
// ===== library: MasterCopy "LSim_AllPass1OrdReal" =====

FUNCTION_BLOCK "LSim_AllPass1OrdReal"   // FB61, SCL
{ S7_Optimized_Access := 'TRUE' }
VERSION : 2.01
   VAR_INPUT
      calcParam : Bool;   // recalculate with new parameters
      input : Real;   // input signal
      tmLag1 : Real := 2.0;   // time constant T1 [sec]
      gain : Real := 1.0;   // gain factor
      cycle : Real := 0.1;   // cyclic time [sec]
      maxOut : Real := 100.0;   // max. output limit
      minOut : Real;   // min. output limit
      reset : Bool;   // resets all relevant parameters to ‘0’ including the output
   END_VAR
   VAR_OUTPUT
      error : Bool;   // error (#tmLag1 <= 0)
      status : Word;   // status (if #tmLag1 <= 0 then status = 16#8001)
      maxReached : Bool;   // output has reached max. limit
      minReached : Bool;   // output has reached min. limit
      output : Real;   // output signal (if #error = FALSE)
   END_VAR
   VAR
      statRxn1 : Real;   // delayed input signal (n-1)
      statRyn1 : Real;   // delayed output signal (n-1)
      statRb1 : Real;
      statRa1 : Real;
      statOutput : Real;   // output signal
   END_VAR
BEGIN
   //=============================================================================
   //SIEMENS AG
   //(c)Copyright 2017 All Rights Reserved
   //-----------------------------------------------------------------------------
   //Library:       Library for Controlled System Simulation
   //Tested with:   S7-1500 FW V2.0 / S7-1200 FW V4.2
   //Engineering:   STEP 7 V14 Upd2 (TIA Portal)
   //Restrictions:  Cyclic interrupt
   //Requirements:  memory card needed for S7-1500
   //Functionality: Simulation of an All-Pass 1. Order with real p-Poles
   //
   //         gain * (1 - tmLag1*p)
   //  F(p) = ---------------------
   //            (1 + tmLag1*p)
   //          
   //  Call the simulation in a cyclic interrupt with
   //  cyclic interrupt time at least = tmLag1/10!
   //-----------------------------------------------------------------------------
   //Change log table:
   //Version  Date       Expert in charge                Changes applied
   //02.00.00 03.02.2016 Siemens Industry Online Support Release (STEP 7 V13 SP1)
   //02.00.01 02.03.2017 Siemens Industry Online Support Release (STEP 7 V14)
   //=============================================================================

   // check of the parameter
   IF #tmLag1 <= 0 THEN
     #error := True;
     #status := W#16#8001;     // Parameter Error
     #statRxn1 := 0.0;
     #statRyn1 := 0.0;
     #statOutput := 0;
     #output := 0;
     RETURN;
   ELSE
     #error := FALSE;
     #status := W#16#0000;     // no error
   END_IF;


   // Z-parameters 
   IF #calcParam = True THEN
   // Calculate z-parameters for allpass filter
      #statRa1 := -EXP(-#cycle/#tmLag1);
      #statRb1 := #gain*(2 + #statRa1);

   END_IF;
   // reset Memory
   IF #reset = True THEN
     #statRxn1 := 0.0;
     #statRyn1 := 0.0;
     #statOutput:=0;
     #error := False;
     #status := W#16#0000;
   END_IF;

   // save delayed output signal 
   #statRyn1:= #statOutput;

   // Differencial Equation of all-pass filter 1. order
   #statOutput := #input * (-#gain) +  #statRxn1* #statRb1 - #statRyn1*#statRa1;

   // save delayed input signals
   #statRxn1 := #input;

   // max limit of acutating variable
   IF #statOutput > #maxOut THEN
     #statOutput := #maxOut;
     #maxReached:= True;
   ELSE
     #maxReached := False;
   END_IF;

   // min limit of acutating variable
   IF #statOutput < #minOut THEN
     #statOutput := #minOut;
     #minReached := True;
   ELSE
     #minReached := False;
   END_IF;

   #output := #statOutput;
END_FUNCTION_BLOCK

// ===== library: MasterCopy "LSim_AllPass2OrdReal" =====

FUNCTION_BLOCK "LSim_AllPass2OrdReal"   // FB62, SCL
{ S7_Optimized_Access := 'TRUE' }
VERSION : 2.01
   VAR_INPUT
      calcParam : Bool;   // recalculate with new parameters
      input : Real;   // input signal
      tmLag1 : Real := 2.0;   // time constant T1 [sec]
      tmLag2 : Real := 0.2;   // time constant T2 [sec]
      gain : Real := 1.0;   // gain factor
      cycle : Real := 0.1;   // cyclic time [sec]
      maxOut : Real := 100.0;   // max. output limit
      minOut : Real;   // min. output limit
      reset : Bool;   // resets all relevant parameters to ‘0’ including the output
   END_VAR
   VAR_OUTPUT
      error : Bool;   // error (#tmLag1 <= 0 or #tmLag2 <= 0 or #tmLag2 = #tmLag1)
      status : Word;   // status (if #error = TRUE then status = 16#8001)
      maxReached : Bool;   // output has reached max. limit
      minReached : Bool;   // output has reached min. limit
      output : Real;   // output signal (if #error = FALSE)
   END_VAR
   VAR
      statRxn2 : Real;   // delayed input signal (n-2)
      statRxn1 : Real;   // delayed input signal (n-1)
      statRyn2 : Real;   // delayed output signal (n-2)
      statRyn1 : Real;   // delayed output signal (n-1)
      statRb1 : Real;
      statRb2 : Real;
      statRa1 : Real;
      statRa2 : Real;
      statRe1 : Real;
      statRe2 : Real;
      statRk1 : Real;
      statOverfirst : Bool;
      statOutput : Real;   // output signal
   END_VAR
BEGIN
   //=============================================================================
   //SIEMENS AG
   //(c)Copyright 2017 All Rights Reserved
   //-----------------------------------------------------------------------------
   //Library:       Library for Controlled System Simulation
   //Tested with:   S7-1500 FW V2.0 / S7-1200 FW V4.2
   //Engineering:   STEP 7 V14 Upd2 (TIA Portal)
   //Restrictions:  Cyclic interrupt
   //Requirements:  memory card needed for S7-1500
   //Functionality: Simulation of an All-Pass 2. Order with real p-Poles
   //
   //         gain * (1 - tmLag1*p) * (1 - tmLag2*p)
   //  F(p) = --------------------------------------
   //            (1 + tmLag1*p) * (1 + tmLag2*p)
   //          
   //  Call the simulation in a cyclic interrupt with
   //  cyclic interrupt time at least = tmLag1/10!
   //-----------------------------------------------------------------------------
   //Change log table:
   //Version  Date       Expert in charge                Changes applied
   //02.00.00 03.02.2016 Siemens Industry Online Support Release (STEP 7 V13 SP1)
   //02.00.01 02.03.2017 Siemens Industry Online Support Release (STEP 7 V14)
   //=============================================================================

   // check of the parameter
   IF #tmLag1 <= 0 OR #tmLag2 <= 0 OR #tmLag1 = #tmLag2 THEN
     #error := TRUE;
     #status := W#16#8001;     // Parameter Error
     #statRxn1 := 0.0;
     #statRyn1 := 0.0;
     #statRxn2 := 0.0;
     #statRyn2 := 0.0;
     #statOutput := 0;
     #output := 0;
     RETURN;
   ELSE
     #error := FALSE;
     #status := W#16#0000;     // no error
   END_IF;

   // calculates the z-parameter for the difference equatation
   IF #calcParam = True OR NOT #statOverfirst THEN
   // Calculate z-parameters for oscilating PT2-System
   #statOverfirst:=1;
   #statRe1 := -EXP(-#cycle/#tmLag1);
   #statRe2 := -EXP(-#cycle/#tmLag2);
   #statRk1 := (2* (#tmLag2 + #tmLag1))/(#tmLag2 - #tmLag1);
   #statRa1 := #statRe1 + #statRe2;
   #statRa2 := #statRe1*#statRe2;
   #statRb1 := #gain*(#statRa1+ #statRk1*(#statRe2 - #statRe1));
   #statRb2 := #gain*(#statRa2 -#statRk1*(#statRe2 - #statRe1));
   END_IF;

   // reset memory
   IF #reset = True THEN
     #statRxn1 := 0.0;
     #statRyn1 := 0.0;
     #statRxn2 := 0.0;
     #statRyn2 := 0.0;
     #statOutput:=0;
     #error := False;
     #status := W#16#0000;
   END_IF;

   // save delayed output-signals
   #statRyn2:=#statRyn1;
   #statRyn1:= #statOutput;

   // difference equatation for PT2-system
   #statOutput := #input * #gain +  #statRxn1* #statRb1 + #statRxn2*#statRb2 - #statRyn1*#statRa1 - #statRyn2*#statRa2;

   // save delayed input-signals
   #statRxn2 := #statRxn1;
   #statRxn1 := #input;

   // max limit of acutating variable
   IF #statOutput > #maxOut THEN
     #statOutput := #maxOut;
     #maxReached:= True;
   ELSE
     #maxReached := False;
   END_IF;

   // min limit of acutating variable
   IF #statOutput < #minOut THEN
     #statOutput := #minOut;
     #minReached := True;
   ELSE
     #minReached := False;
   END_IF;

   #output := #statOutput;
END_FUNCTION_BLOCK

// ===== library: MasterCopy "LSim_DT1" =====

FUNCTION_BLOCK "LSim_DT1"   // FB60, SCL
{ S7_Optimized_Access := 'TRUE' }
VERSION : 2.01
   VAR_INPUT
      calcParam : Bool;   // recalculate with new parameters
      input : Real;   // input signal
      tmLag1 : Real := 2.0;   // time constant T1 [sec]
      tmLag2 : Real := 0.5;   // time constant T2 [sec]
      gain : Real := 1.0;   // gain factor
      cycle : Real := 0.1;   // cyclic time [sec]
      maxOut : Real := 100.0;   // max. output limit
      minOut : Real := -100.0;   // min. output limit
      reset : Bool;   // resets all relevant parameters to ‘0’ including the output
   END_VAR
   VAR_OUTPUT
      error : Bool;   // error (#tmLag1 <= 0)
      status : Word;   // status (if #tmLag1 <= 0 then status = 16#8001)
      maxReached : Bool;   // output has reached max. limit
      minReached : Bool;   // output has reached min. limit
      output : Real;   // output signal (if #error = FALSE)
   END_VAR
   VAR
      statRxn1 : Real;   // delayed input signal (n-1)
      statRyn1 : Real;   // delayed output signal (n-1)
      statRb0 : Real;
      statRa1 : Real;
      statOverfirst : Bool;
      statOutput : Real;   // output signal
   END_VAR
BEGIN
   //=============================================================================
   //SIEMENS AG
   //(c)Copyright 2017 All Rights Reserved
   //-----------------------------------------------------------------------------
   //Library:       Library for Controlled System Simulation
   //Tested with:   S7-1500 FW V2.0 / S7-1200 FW V4.2
   //Engineering:   STEP 7 V14 Upd2 (TIA Portal)
   //Restrictions:  Cyclic interrupt
   //Requirements:  memory card needed for S7-1500
   //Functionality: Simulation of a DT1-System
   //
   //         gain * tmLag2 * p
   //  F(p) = ------------------------------
   //            (1 + tmLag1*p)
   //          
   //  Call the simulation in a cyclic interrupt with
   //  cyclic interrupt time at least = tmLag1/10!
   //-----------------------------------------------------------------------------
   //Change log table:
   //Version  Date       Expert in charge                Changes applied
   //02.00.00 03.02.2016 Siemens Industry Online Support Release (STEP 7 V13 SP1)
   //02.00.01 02.03.2017 Siemens Industry Online Support Release (STEP 7 V14)
   //=============================================================================

   // check of the parameter
   IF #tmLag1 <= 0 THEN
     #error := true;
     #status := W#16#8001; // parameter error
     #statRxn1 := 0.0;
     #statRyn1 := 0.0;
     #statOutput := 0;
     #output := 0;
     RETURN;
   ELSE
     #error := FALSE;
     #status := W#16#0000;     // no error
   END_IF;

   // calculates the z-parameter for the difference equatation
   IF #calcParam = True OR NOT #statOverfirst THEN 
     // Calculate the z-parameter for the DT1-System
     #statOverfirst := 1;
     #statRa1 := -EXP(-#cycle/#tmLag1);
     #statRb0 := #gain*(#tmLag2/#tmLag1);
   END_IF;

   // reset Memory
   IF #reset = True THEN
     #statRxn1 := 0.0;
     #statRyn1 := 0.0;
     #statOutput:=0;
     #error := false;
     #status := W#16#0000;
   END_IF;

   // save delayed output-signals
   #statRyn1:= #statOutput;

   //  difference equatation for DT1-system
   #statOutput := #input * #statRb0 - #statRxn1* #statRb0 - #statRyn1*#statRa1;

   // save delayed input-signals
   #statRxn1 := #input;

   // max limit of acutating variable
   IF #statOutput > #maxOut THEN
     #statOutput := #maxOut;
     #maxReached := True;
   ELSE
     #maxReached := False;
   END_IF;

   // min limit of acutating variable
   IF #statOutput < #minOut THEN
     #statOutput := #minOut;
     #minReached := True;
   ELSE
     #minReached := False;
   END_IF;

   #output := #statOutput;
END_FUNCTION_BLOCK

// ===== library: MasterCopy "LSim_I" =====

FUNCTION_BLOCK "LSim_I"   // FB56, SCL
{ S7_Optimized_Access := 'TRUE' }
VERSION : 2.01
   VAR_INPUT
      calcParam : Bool;   // recalculate with new parameters
      input : Real;   // input signal
      tmLag1 : Real := 1.0;   // time constant T1 [sec]
      cycle : Real := 0.1;   // cyclic time [sec]
      maxOut : Real := 100.0;   // max. output limit
      minOut : Real;   // min. output limit
      reset : Bool;   // resets all relevant parameters to ‘0’ including the output
   END_VAR
   VAR_OUTPUT
      error : Bool;   // error (#tmLag1 <= 0)
      status : Word;   // status (if #tmLag1 <= 0 then status = 16#8001)
      maxReached : Bool;   // output has reached max. limit
      minReached : Bool;   // output has reached min. limit
      output : Real;   // output signal (if #error = FALSE)
   END_VAR
   VAR
      statRxn1 : Real;   // delayed input signal (n-1)
      statRyn1 : Real;   // delayed output signal (n-1)
      statRa1 : Real;
      statRb1 : Real;
      statOverfirst : Bool;
      statOutput : Real;   // output signal
   END_VAR
BEGIN
   //=============================================================================
   //SIEMENS AG
   //(c)Copyright 2017 All Rights Reserved
   //-----------------------------------------------------------------------------
   //Library:       Library for Controlled System Simulation
   //Tested with:   S7-1500 FW V2.0 / S7-1200 FW V4.2
   //Engineering:   STEP 7 V14 Upd2 (TIA Portal)
   //Restrictions:  Cyclic interrupt
   //Requirements:  memory card needed for S7-1500
   //Functionality: Simulation of a I-System
   //
   //             1
   //  F(p) = -----------
   //         (tmLag1*p)
   //          
   //  Call the simulation in a cyclic interrupt with
   //  cyclic interrupt time at least = tmLag1/10!
   //-----------------------------------------------------------------------------
   //Change log table:
   //Version  Date       Expert in charge                Changes applied
   //02.00.00 03.02.2016 Siemens Industry Online Support Release (STEP 7 V13 SP1)
   //02.00.01 02.03.2017 Siemens Industry Online Support Release (STEP 7 V14)
   //=============================================================================

   // check parameter
   IF #tmLag1 <= 0 THEN
     #error := True;
     #status := W#16#8001;     // Parameter Error
     #statRxn1 := 0.0;
     #statRyn1 := 0.0;
     #statOutput := 0;
     #output := 0;
     RETURN;
   ELSE
     #error := FALSE;
     #status := W#16#0000;     // no error
   END_IF;

   // calculates the z-parameter for the difference equatation
   IF #calcParam = True OR NOT #statOverfirst THEN
   #statOverfirst:=1;
     // Calculate z-parameters for IT1-System
   #statRb1 := #cycle/#tmLag1;
   #statRa1 := -1;

   END_IF;

   // reset Memory
   IF #reset = True THEN
     #statRxn1 := 0.0;
     #statRyn1 := 0.0;
     #statOutput:=0;
   END_IF;

   // save delayed output-signals
   #statRyn1:= #statOutput;

   // difference equatation for the I-system
   #statOutput := #statRxn1* #statRb1 - #statRyn1*#statRa1;

   // save delayed input-signals
   #statRxn1 := #input;

   // max limit of acutating variable
   IF #statOutput > #maxOut THEN
     #statOutput := #maxOut;
     #maxReached:= True;
   ELSE
     #maxReached := False;
   END_IF;

   // min limit of acutating variable
   IF #statOutput < #minOut THEN
     #statOutput := #minOut;
     #minReached := True;
   ELSE
     #minReached := False;
   END_IF;

   #output := #statOutput;
END_FUNCTION_BLOCK

// ===== library: MasterCopy "LSim_IT1" =====

FUNCTION_BLOCK "LSim_IT1"   // FB57, SCL
{ S7_Optimized_Access := 'TRUE' }
VERSION : 2.01
   VAR_INPUT
      calcParam : Bool;   // recalculate with new parameters
      input : Real;   // input signal
      tmLag1 : Real := 5.0;   // time constant T1 [sec]
      gain : Real := 1.0;   // gain factor
      cycle : Real := 0.1;   // cyclic time [sec]
      maxOut : Real := 100.0;   // max. output limit
      minOut : Real;   // min. output limit
      reset : Bool;   // resets all relevant parameters to ‘0’ including the output
   END_VAR
   VAR_OUTPUT
      error : Bool;   // error (#tmLag1 <= 0)
      status : Word;   // status (if #tmLag1 <= 0 then status = 16#8001)
      maxReached : Bool;   // output has reached max. limit
      minReached : Bool;   // output has reached min. limit
      output : Real;   // output signal (if #error = FALSE)
   END_VAR
   VAR
      statRxn2 : Real;   // delayed input signal (n-2)
      statRxn1 : Real;   // delayed input signal (n-1)
      statRyn2 : Real;   // delayed output signal (n-2)
      statRyn1 : Real;   // delayed output signal (n-1)
      statRf1 : Real;
      statRf2 : Real;
      statRe1 : Real;
      statRe2 : Real;
      statAlpha : Real;
      statOverfirst : Bool;
      statOutput : Real;   // output signal
   END_VAR
BEGIN
   //=============================================================================
   //SIEMENS AG
   //(c)Copyright 2017 All Rights Reserved
   //-----------------------------------------------------------------------------
   //Library:       Library for Controlled System Simulation
   //Tested with:   S7-1500 FW V2.0 / S7-1200 FW V4.2
   //Engineering:   STEP 7 V14 Upd2 (TIA Portal)
   //Restrictions:  Cyclic interrupt
   //Requirements:  memory card needed for S7-1500
   //Functionality: Simulation of a IT1-System
   //  
   //               gain
   //  F(p) = ------------------
   //         p * (tmLag1*p + 1)
   //         
   //  Call the simulation in a cyclic interrupt with
   //  cyclic interrupt time at least = tmLag1/10!
   //-----------------------------------------------------------------------------
   //Change log table:
   //Version  Date       Expert in charge                Changes applied
   //02.00.00 03.02.2016 Siemens Industry Online Support Release (STEP 7 V13 SP1)
   //02.00.01 02.03.2017 Siemens Industry Online Support Release (STEP 7 V14)
   //=============================================================================


   // check parameter
   IF #tmLag1 <= 0 THEN
     #error := True;
     #status := W#16#8001;     // Parameter Error
     #statRxn1 := 0.0;
     #statRyn1 := 0.0;
     #statRxn2 := 0.0;
     #statRyn2 := 0.0;
     #statOutput := 0;
     #output := 0;
     RETURN;
   ELSE
     #error := FALSE;
     #status := W#16#0000;     // no error
   END_IF;

   // calculates the z-parameter for the difference equatation
   IF #calcParam = True OR NOT #statOverfirst THEN
     #statOverfirst:=1;
   // calculates the z-parameter for the difference equatation of the IT1-System
   #statAlpha := EXP(-#cycle/#tmLag1);
   #statRe1 := -1 - #statAlpha;
   #statRe2 := #statAlpha;
   #statRf1 := #gain*(#cycle +(#statAlpha - 1)*#tmLag1);
   #statRf2 := #gain*(-#statAlpha*#cycle+(1-#statAlpha)*#tmLag1);
   END_IF;

   // reset Memory
   IF #reset = True THEN
     #statRxn1 := 0.0;
     #statRyn1 := 0.0;
     #statRxn2 := 0.0;
     #statRyn2 := 0.0;
     #statOutput:=0;
   END_IF;

   // save delayed output-signals
   #statRyn2:=#statRyn1;
   #statRyn1:= #statOutput;

   // difference equatation for IT1-System
   #statOutput := #statRxn1* #statRf1 + #statRxn2*#statRf2 - #statRyn1*#statRe1 - #statRyn2*#statRe2;

   // save delayed input-signals
   #statRxn2 := #statRxn1;
   #statRxn1 := #input;

   // max limit of acutating variable
   IF #statOutput > #maxOut THEN
   #statOutput := #maxOut;
   #maxReached := True;
   ELSE
     #maxReached := False;
   END_IF;

   // min limit of acutating variable
   IF #statOutput < #minOut THEN
     #statOutput := #minOut;
     #minReached := True;
   ELSE
     #minReached := False;
   END_IF;

   #output := #statOutput;
END_FUNCTION_BLOCK

// ===== library: MasterCopy "LSim_Lagging" =====

FUNCTION_BLOCK "LSim_Lagging"   // FB59, SCL
{ S7_Optimized_Access := 'TRUE' }
VERSION : 2.02
   VAR_INPUT
      input : Real;   // input signal
   END_VAR
   VAR_OUTPUT
      output : Real;   // output signal
   END_VAR
   VAR_IN_OUT
      delayCycles : UInt;   // number of cycles the input signal is delayed (if #delayCycles > #MAX then #delayCycles = #MAX)
   END_VAR
   VAR
      statDelayStore : Array[0..#MAX] of Real;
      statIndexRead : Int;
      statIndexWrite : Int;
   END_VAR
   VAR CONSTANT
      MAX : Int := 100;   // maximum size of array #statDelayStore
   END_VAR
BEGIN
   //=============================================================================
   //SIEMENS AG
   //(c)Copyright 2017 All Rights Reserved
   //-----------------------------------------------------------------------------
   //Library:       Library for Controlled System Simulation
   //Tested with:   S7-1500 FW V2.0 / S7-1200 FW V4.2
   //Engineering:   STEP 7 V14 Upd2 (TIA Portal)
   //Restrictions:  Cyclic interrupt
   //Requirements:  memory card needed for S7-1500
   //Functionality: Simulation of an Tt-System (Lagging)
   //
   //  F(p) = EXP(-p * delayCycles * cyclic interrupt time)
   //          
   //  Call the simulation in a cyclic interrupt with
   //  cyclic interrupt time at least = tmLag1/10!
   //-----------------------------------------------------------------------------
   //Change log table:
   //Version  Date       Expert in charge                Changes applied
   //02.00.00 03.02.2016 Siemens Industry Online Support Release (STEP 7 V13 SP1)
   //02.00.01 02.03.2017 Siemens Industry Online Support Optimize program code
   //02.00.02 02.03.2017 Siemens Industry Online Support Release (STEP 7 V14)
   //=============================================================================

   // Check Parameters
   IF #delayCycles > #MAX THEN
     #delayCycles := INT_TO_UINT(#MAX);
   ELSE
     #delayCycles := #delayCycles;
   END_IF;

   IF #statIndexWrite < #delayCycles THEN
     #statDelayStore[#statIndexWrite] := #input;   // write input at delayStore indexWrite
     #statIndexRead := #statIndexWrite + 1;
     #output := #statDelayStore[#statIndexRead];   // read output from delayStore indexWrite + 1
     #statIndexWrite := #statIndexWrite + 1;       // increment delayStore indexWrite
   ELSE // maximum reached
     #statDelayStore[#statIndexWrite] := #input;   // write input at delayStore maximum
     #statIndexRead := 0;                          // set indexRead to beginning
     #output := #statDelayStore[#statIndexRead];   // read output from delayStore indexRead
     #statIndexWrite := 0;                         // set indexWrite to beginning
   END_IF;
END_FUNCTION_BLOCK

// ===== library: MasterCopy "LSim_PDT1" =====

FUNCTION_BLOCK "LSim_PDT1"   // FB55, SCL
{ S7_Optimized_Access := 'TRUE' }
VERSION : 2.01
   VAR_INPUT
      calcParam : Bool;   // recalculate with new parameters
      input : Real;   // input signal
      tmLag1 : Real := 2.0;   // time constant T1 [sec]
      tmLag2 : Real := 0.2;   // time constant T2 [sec]
      gain : Real := 1.0;   // gain factor
      cycle : Real := 0.1;   // cyclic time [sec]
      maxOut : Real := 100.0;   // max. output limit
      minOut : Real;   // min. output limit
      reset : Bool;   // resets all relevant parameters to ‘0’ including the output
   END_VAR
   VAR_OUTPUT
      error : Bool;   // error (#tmLag1 <= 0 or #tmLag2 <= 0)
      status : Word;   // status (if #error = TRUE then status = 16#8001)
      maxReached : Bool;   // output has reached max. limit
      minReached : Bool;   // output has reached min. limit
      output : Real;   // output signal (if #error = FALSE)
   END_VAR
   VAR
      statRxn2 : Real;   // delayed input signal (n-2)
      statRxn1 : Real;   // delayed input signal (n-1)
      statRyn2 : Real;   // delayed output signal (n-2)
      statRyn1 : Real;   // delayed output signal (n-1)
      statRb1 : Real;
      statRb0 : Real;
      statRa1 : Real;
      statOverfirst : Bool;
      statOutput : Real;
   END_VAR
BEGIN
   //=============================================================================
   //SIEMENS AG
   //(c)Copyright 2017 All Rights Reserved
   //-----------------------------------------------------------------------------
   //Library:       Library for Controlled System Simulation
   //Tested with:   S7-1500 FW V2.0 / S7-1200 FW V4.2
   //Engineering:   STEP 7 V14 Upd2 (TIA Portal)
   //Restrictions:  Cyclic interrupt
   //Requirements:  memory card needed for S7-1500
   //Functionality: Simulation of an PD-T1 System
   //
   //         gain * (1 + tmLag2*p)
   //  F(p) = ------------------------------
   //            (1 + tmLag1*p)
   //          
   //  Call the simulation in a cyclic interrupt with
   //  cyclic interrupt time at least = tmLag1/10!
   //-----------------------------------------------------------------------------
   //Change log table:
   //Version  Date       Expert in charge                Changes applied
   //02.00.00 03.02.2016 Siemens Industry Online Support Release (STEP 7 V13 SP1)
   //02.00.01 02.03.2017 Siemens Industry Online Support Release (STEP 7 V14)
   //=============================================================================

   // check parameter
   IF #tmLag1 <= 0 OR #tmLag2 <= 0 THEN
     #error := True;
     #status := W#16#8001;     // Parameter Error
     #statRxn1 := 0.0;
     #statRyn1 := 0.0;
     #statRxn2 := 0.0;
     #statRyn2 := 0.0;
     #statOutput := 0;
     #output := 0;
     RETURN;
   ELSE
     #error := FALSE;
     #status := W#16#0000;     // no error
   END_IF;

   // calculates the z-parameter for the difference equatation
   IF #calcParam = True OR NOT #statOverfirst THEN
     #statOverfirst := 1;
   // Calculate z-parameters for oscilating PT2-System
   #statRa1 := -EXP(-#cycle/#tmLag1);
   #statRb0 := #gain *(#tmLag2/#tmLag1);
   #statRb1 := #gain *(1 + #statRa1 - (#tmLag2/#tmLag1));
   END_IF;

   // reset Memory
   IF #reset = True THEN
     #statRxn1 := 0.0;
     #statRyn1 := 0.0;
     #statRxn2 := 0.0;
     #statRyn2 := 0.0;
     #statOutput:=0;
     #error := False;
     #status := W#16#0000;
   END_IF;

   // save delayed output-signals
   #statRyn1:= #statOutput;

   // difference equatation for PT2-system
   #statOutput := #input * #statRb0 +  #statRxn1* #statRb1 - #statRyn1*#statRa1;

   // save delayed input-signals
   #statRxn1 := #input;

   // max limit of acutating variable
   IF #statOutput > #maxOut THEN
     #statOutput := #maxOut;
     #maxReached:= True;
   ELSE
     #maxReached := False;
   END_IF;

   // min limit of acutating variable
   IF #statOutput < #minOut THEN
     #statOutput := #minOut;
     #minReached := True;
   ELSE
     #minReached := False;
   END_IF;

   #output := #statOutput;
END_FUNCTION_BLOCK

// ===== library: MasterCopy "LSim_PT1" =====

FUNCTION_BLOCK "LSim_PT1"   // FB50, SCL
{ S7_Optimized_Access := 'TRUE' }
VERSION : 2.01
   VAR_INPUT
      calcParam : Bool;   // recalculate with new parameters
      input : Real;   // input signal
      tmLag1 : Real := 1.0;   // time constant T1 [sec]
      gain : Real := 1.0;   // gain factor
      cycle : Real := 0.1;   // cyclic time [sec]
      maxOut : Real := 100.0;   // max. output limit
      minOut : Real;   // min. output limit
      reset : Bool;   // resets all relevant parameters to ‘0’ including the output
   END_VAR
   VAR_OUTPUT
      error : Bool;   // error (#tmLag1 <= 0)
      status : Word;   // status (if #tmLag1 <= 0 then status = 16#8001)
      maxReached : Bool;   // output has reached max. limit
      minReached : Bool;   // output has reached min. limit
      output : Real;   // output signal (if #error = FALSE)
   END_VAR
   VAR
      statRf1 : Real;
      statRe1 : Real;
      statOverfirst : Bool;
      statOutput : Real;
   END_VAR
BEGIN
   //=============================================================================
   //SIEMENS AG
   //(c)Copyright 2017 All Rights Reserved
   //-----------------------------------------------------------------------------
   //Library:       Library for Controlled System Simulation
   //Tested with:   S7-1500 FW V2.0 / S7-1200 FW V4.2
   //Engineering:   STEP 7 V14 Upd2 (TIA Portal)
   //Restrictions:  Cyclic interrupt
   //Requirements:  memory card needed for S7-1500
   //Functionality: Simulation of a PT1-System
   //
   //              gain
   //  F(p) = ---------------
   //          tmLag1 * p + 1
   //          
   //  Call the simulation in a cyclic interrupt with
   //  cyclic interrupt time at least = tmLag1/10!
   //-----------------------------------------------------------------------------
   //Change log table:
   //Version  Date       Expert in charge                Changes applied
   //02.00.00 03.02.2016 Siemens Industry Online Support Release (STEP 7 V13 SP1)
   //02.00.01 02.03.2017 Siemens Industry Online Support Release (STEP 7 V14)
   //=============================================================================
   // check parameter
   IF #tmLag1 <= 0 THEN
     #error := TRUE;
     #status := W#16#8001;     // Parameter Error
     #statOutput := 0;
     #output := 0;
     RETURN;
   ELSE
     #error := FALSE;
     #status := W#16#0000;     // no error
   END_IF;

   IF #calcParam = True OR NOT #statOverfirst THEN
     #statOverfirst:=1;
   // Z-parameters For Laplace PT1-System
   #statRe1 := - EXP(-#cycle/#tmLag1);
   #statRf1 := #gain*(1 + #statRe1);
   END_IF;

   // Differencial Equation of PT1-System
   #statOutput := #input*#statRf1 - #statOutput*#statRe1;

   // max limit of acutating variable
   IF #statOutput > #maxOut THEN
     #statOutput := #maxOut;
     #maxReached:= True;
   ELSE
     #maxReached := False;
   END_IF;

   // min limit of acutating variable
   IF #statOutput < #minOut THEN
     #statOutput := #minOut;
     #minReached := True;
   ELSE
     #minReached := False;
   END_IF;

   IF #reset THEN
     #statOutput := 0;
   END_IF;

   #output := #statOutput;
END_FUNCTION_BLOCK

// ===== library: MasterCopy "LSim_PT1asym" =====

FUNCTION_BLOCK "LSim_PT1asym"   // FB51, SCL
{ S7_Optimized_Access := 'TRUE' }
VERSION : 2.01
   VAR_INPUT
      calcParam : Bool;   // recalculate with new parameters
      input : Real;   // input signal
      tmLag1up : Real := 1.0;   // time constant T1 [sec] rising input
      tmLag1down : Real := 10.0;   // time constant T1 [sec] falling input
      gain : Real := 1.0;   // gain factor
      cycle : Real := 0.1;   // cyclic time [sec]
      maxOut : Real := 100.0;   // max. output limit
      minOut : Real;   // min. output limit
      reset : Bool;   // resets all relevant parameters to ‘0’ including the output
   END_VAR
   VAR_OUTPUT
      error : Bool;   // error (#tmLag1 <= 0 or #tmLag2 <= 0)
      status : Word;   // status (if #error = TRUE then status = 16#8001)
      maxReached : Bool;   // output has reached max. limit
      minReached : Bool;   // output has reached min. limit
      output : Real;   // output signal (if #error = FALSE)
   END_VAR
   VAR
      statRxn1 : Real;   // delayed input signal (n-1)
      statRyn1 : Real;   // delayed output signal (n-1)
      statRf1up : Real;   // Z-parameter 1 (rising xn)
      statRe1up : Real;   // Z-parameter 2 (rising xn)
      statRf1dn : Real;   // Z-parameter 1 (falling xn)
      statRe1dn : Real;   // Z-parameter 2 (falling xn)
      statRf1 : Real;   // active Z-parameter 1
      statRe1 : Real;   // active Z-parameter 2
      statOverfirst : Bool;
      statOutput : Real;
   END_VAR
BEGIN
   //=============================================================================
   //SIEMENS AG
   //(c)Copyright 2017 All Rights Reserved
   //-----------------------------------------------------------------------------
   //Library:       Library for Controlled System Simulation
   //Tested with:   S7-1500 FW V2.0 / S7-1200 FW V4.2
   //Engineering:   STEP 7 V14 Upd2 (TIA Portal)
   //Restrictions:  Cyclic interrupt
   //Requirements:  memory card needed for S7-1500
   //Functionality: Simulation of a PT1-System with two different Time-Constants
   //
   //  tmLag1up: Time-Constant for positive Inputsignal changes 
   //  tmLag1down: Time-Constant for negative Inputsignal changes
   //  
   //                gain
   //  Fup(p) = ----------------
   //           tmLag1up * p + 1
   //          
   //                    gain
   //  Fdown(p) = ------------------
   //             tmLag1down * p + 1
   //          
   //  Call the simulation in a cyclic interrupt with
   //  //  cyclic interrupt time at least = tmLag1/10!
   //-----------------------------------------------------------------------------
   //Change log table:
   //Version  Date       Expert in charge                Changes applied
   //02.00.00 03.02.2016 Siemens Industry Online Support Release (STEP 7 V13 SP1)
   //02.00.01 02.03.2017 Siemens Industry Online Support Release (STEP 7 V14)
   //=============================================================================

   // check parameter
   IF #tmLag1up <= 0 OR #tmLag1down <= 0 THEN
     #error := TRUE;
     #status := W#16#8001;     // Parameter Error
     #statOutput := 0;
     #output := 0;
     RETURN;
   ELSE
     #error := FALSE;
     #status := W#16#0000;     // no error
   END_IF;

   IF #calcParam = True OR NOT #statOverfirst THEN
     #statOverfirst:=1;
   // Z-parameters for Laplace PT1-System (rising signal change)
   #statRe1up := - EXP(-#cycle/#tmLag1up);
   #statRf1up := #gain*(1 + #statRe1up);
   // Z-parameters for Laplace PT1-System (falling signal change)
   #statRe1dn := - EXP(-#cycle/#tmLag1down);
   #statRf1dn := #gain*(1 + #statRe1dn);
   END_IF;

   // save delayed output signals
   #statRyn1:= #statOutput;

   // Change the parameter sets, dependent to Input Change
   IF (#input - #statRxn1) > 0 THEN
     #statRf1 := #statRf1up;
     #statRe1 := #statRe1up;
   ELSIF (#input - #statRxn1) < 0 THEN
      #statRf1 := #statRf1dn;
      #statRe1 := #statRe1dn;
   ELSE
     ;
   END_IF;

   // Differencial Equation of PT1-System
   #statOutput := #input*#statRf1 - #statRyn1*#statRe1;

   // save delayed input signals
   #statRxn1 := #input;

   // max limit of acutating variable
   IF #statOutput > #maxOut THEN
     #statOutput := #maxOut;
     #maxReached:= True;
   ELSE
     #maxReached := False;
   END_IF;

   // min limit of acutating variable
   IF #statOutput < #minOut THEN
     #statOutput := #minOut;
     #minReached := True;
   ELSE
     #minReached := False;
   END_IF;

   IF #reset THEN
     #statOutput := 0;
   END_IF;

   #output := #statOutput;
END_FUNCTION_BLOCK

// ===== library: MasterCopy "LSim_PT2aper" =====

FUNCTION_BLOCK "LSim_PT2aper"   // FB53, SCL
{ S7_Optimized_Access := 'TRUE' }
VERSION : 2.01
   VAR_INPUT
      calcParam : Bool;   // recalculate with new parameters
      input : Real;   // input signal
      tmLag1 : Real := 2.0;   // time constant T1 [sec]
      tmLag2 : Real := 0.2;   // time constant T2 [sec]
      gain : Real := 1.0;   // gain factor
      cycle : Real := 0.1;   // cyclic time [sec]
      maxOut : Real := 100.0;   // max. output limit
      minOut : Real;   // min. output limit
      reset : Bool;   // resets all relevant parameters to ‘0’ including the output
   END_VAR
   VAR_OUTPUT
      error : Bool;   // error (#tmLag1 <= 0 or #tmLag2 <= 0 or #tmLag1 = #tmLag2)
      status : Word;   // status (if #error = TRUE then status = 16#8001)
      maxReached : Bool;   // output has reached max. limit
      minReached : Bool;   // output has reached min. limit
      output : Real;   // output signal (if #error = FALSE)
   END_VAR
   VAR
      statRxn2 : Real;   // delayed input signal (n-2)
      statRxn1 : Real;   // delayed input signal (n-1)
      statRyn2 : Real;   // delayed output signal (n-2)
      statRyn1 : Real;   // delayed output signal (n-1)
      statRf1 : Real;
      statRf2 : Real;
      statRe1 : Real;
      statRe2 : Real;
      statAlpha : Real;
      statBeta : Real;
      statGamma : Real;
      statDelta : Real;
      statOverfirst : Bool;
      statOutput : Real;   // Output signal
   END_VAR
BEGIN
   //=============================================================================
   //SIEMENS AG
   //(c)Copyright 2017 All Rights Reserved
   //-----------------------------------------------------------------------------
   //Library:       Library for Controlled System Simulation
   //Tested with:   S7-1500 FW V2.0 / S7-1200 FW V4.2
   //Engineering:   STEP 7 V14 Upd2 (TIA Portal)
   //Restrictions:  Cyclic interrupt
   //Requirements:  memory card needed for S7-1500
   //Functionality: Simulation of a aperiodic PT2-System
   //  
   //                    gain
   //  F(p) = -----------------------------
   //         (tmLag1*p + 1)*(tmLag2*p + 1)
   //         
   //  Call the simulation in a cyclic interrupt with
   //  cyclic interrupt time at least = tmLag1/10!
   //-----------------------------------------------------------------------------
   //Change log table:
   //Version  Date       Expert in charge                Changes applied
   //02.00.00 03.02.2016 Siemens Industry Online Support Release (STEP 7 V13 SP1)
   //02.00.01 02.03.2017 Siemens Industry Online Support Release (STEP 7 V14)
   //=============================================================================

   // check parameter
   IF #tmLag1 <= 0 OR #tmLag2 <= 0 OR #tmLag1 = #tmLag2 THEN
     #error := TRUE;
     #status := W#16#8001;     // Parameter Error
     #statRxn1 := 0.0;
     #statRyn1 := 0.0;
     #statRxn2 := 0.0;
     #statRyn2 := 0.0;
     #statOutput := 0;
     #output := 0;
     RETURN;
   ELSE
     #error := FALSE;
     #status := W#16#0000;     // no error
   END_IF;

   // calculates the z-parameter for the difference equatation
   IF #calcParam = True OR NOT #statOverfirst THEN
     #statOverfirst := 1;
     // Calculate z-parameters for IT1-System
     #statAlpha := EXP(- #cycle / #tmLag1);
     #statBeta := EXP(- #cycle / #tmLag2);
     #statGamma := #tmLag1 / (#tmLag1 - #tmLag2);
     #statDelta := #tmLag2 / (#tmLag1 - #tmLag2);
     #statRe1 := - #statAlpha - #statBeta;
     #statRe2 := #statAlpha * #statBeta;
     #statRf1 := #gain * (1 - #statGamma * #statAlpha + #statDelta * #statBeta);
     #statRf2 := #gain * (#statAlpha * #statBeta - #statGamma * #statBeta + #statAlpha * #statDelta);
   END_IF;

   // reset Memory
   IF #reset = True THEN
     #statRxn1 := 0.0;
     #statRyn1 := 0.0;
     #statRxn2 := 0.0;
     #statRyn2 := 0.0;
     #statOutput := 0;
   END_IF;
   //save delayed input signals
   #statRxn2 := #statRxn1;
   #statRxn1 := #input;

   //save delayed output signals
   #statRyn2:=#statRyn1;
   #statRyn1:= #statOutput;

   // difference equatation of the PT2-System
   #statOutput := #statRxn1* #statRf1 + #statRxn2*#statRf2 - #statRyn1*#statRe1 - #statRyn2*#statRe2;

   // max limit of acutating variable
   IF #statOutput > #maxOut THEN
     #statOutput := #maxOut;
     #maxReached:= True;
   ELSE
     #maxReached := False;
   END_IF;

   // min limit of acutating variable
   IF #statOutput < #minOut THEN
     #statOutput := #minOut;
     #minReached := True;
   ELSE
     #minReached := False;
   END_IF;

   #output := #statOutput;
END_FUNCTION_BLOCK

// ===== library: MasterCopy "LSim_PT2osc" =====

FUNCTION_BLOCK "LSim_PT2osc"   // FB52, SCL
{ S7_Optimized_Access := 'TRUE' }
VERSION : 2.01
   VAR_INPUT
      calcParam : Bool;   // recalculate with new parameters
      input : Real;   // input signal
      omega : Real := 2.0;   // angular frequency of the undampened vibrations [1/sec]
      damp : Real := 0.2;   // damping (0 < D < 1)
      gain : Real := 1.0;   // gain factor
      cycle : Real := 0.1;   // cyclic time [sec]
      maxOut : Real := 100.0;   // max. output limit
      minOut : Real;   // min. output limit
      reset : Bool;   // resets all relevant parameters to ‘0’ including the output
   END_VAR
   VAR_OUTPUT
      error : Bool;   // error (0 >= damp >= 1 or #omega <= 0)
      status : Word;   // status (if #error = TRUE then status = 16#8001)
      maxReached : Bool;   // output has reached max. limit
      minReached : Bool;   // output has reached min. limit
      output : Real;   // output signal (if #error = FALSE)
   END_VAR
   VAR
      statRxn2 : Real;   // delayed input signal (n-2)
      statRxn1 : Real;   // delayed input signal (n-1)
      statRyn2 : Real;   // delayed output signal (n-2)
      statRyn1 : Real;   // delayed output signal (n-1)
      statRb1 : Real;
      statRb2 : Real;
      statRa1 : Real;
      statRa2 : Real;
      statRo : Real;
      statSigma : Real;
      statNue : Real;
      statOverfirst : Bool;
      statOutput : Real;
   END_VAR
BEGIN
   //=============================================================================
   //SIEMENS AG
   //(c)Copyright 2017 All Rights Reserved
   //-----------------------------------------------------------------------------
   //Library:       Library for Controlled System Simulation
   //Tested with:   S7-1500 FW V2.0 / S7-1200 FW V4.2
   //Engineering:   STEP 7 V14 Upd2 (TIA Portal)
   //Restrictions:  Cyclic interrupt
   //Requirements:  memory card needed for S7-1500
   //Functionality: Simulation of a vibrating PT2-System
   //
   //                  gain
   //  F(p) = ----------------------------------
   //         SQR(p/omega) + 2*damp*p/omega + 1
   //          
   //  Call the simulation in a cyclic interrupt with
   //  cyclic interrupt time at least = tmLag1/10!
   //-----------------------------------------------------------------------------
   //Change log table:
   //Version  Date       Expert in charge                Changes applied
   //02.00.00 03.02.2016 Siemens Industry Online Support Release (STEP 7 V13 SP1)
   //02.00.01 02.03.2017 Siemens Industry Online Support Release (STEP 7 V14)
   //=============================================================================

   // check parameter
   IF #damp >= 1 OR #damp <= 0 OR #omega <= 0 THEN
     #error := TRUE;
     #status := W#16#8001;
     #statRxn1 := 0.0;
     #statRyn1 := 0.0;
     #statRxn2 := 0.0;
     #statRyn2 := 0.0;
     #statOutput := 0;
     #output := 0;
     RETURN;
   ELSE
     #error := FALSE;
     #status := W#16#0000;     // no error 
   END_IF;

   // calculates the z-parameter for the difference equatation
   IF #calcParam = True THEN
   // Calculate z-parameters for oscillating PT2-System
   #statRo := EXP(-2*#omega*#damp*#cycle);
   #statSigma := (COS(#omega * #cycle * SQRT(1 - SQR(#damp)))) * EXP(-#damp*#omega*#cycle);
   #statNue := (SIN(#omega*#cycle*SQRT(1-SQR(#damp)))) * (EXP(-#damp*#omega*#cycle)) * (#damp / SQRT(1 - SQR(#damp)));
   #statRa1 := -2*#statSigma;
   #statRa2 := #statRo;
   #statRb1 := #gain*(1 - #statSigma - #statNue);
   #statRb2 := #gain*(#statRo - #statSigma + #statNue);
   END_IF;

   // reset Memory
   IF #reset = True THEN
     #statRxn1 := 0.0;
     #statRyn1 := 0.0;
     #statRxn2 := 0.0;
     #statRyn2 := 0.0;
     #statOutput:=0;
     #error := False;
     #status := W#16#0000;
   END_IF;

   // save delayed output signals
   #statRyn2:=#statRyn1;
   #statRyn1:= #statOutput;

   // difference equatation for PT2-System
   #statOutput := #statRxn1* #statRb1 + #statRxn2*#statRb2 - #statRyn1*#statRa1 - #statRyn2*#statRa2;

   // save delayed input signals
   #statRxn2 := #statRxn1;
   #statRxn1 := #input;

   // max limit of acutating variable
   IF #statOutput > #maxOut THEN
     #statOutput := #maxOut;
     #maxReached:= True;
   ELSE
     #maxReached := False;
   END_IF;

   // min limit of acutating variable
   IF #statOutput < #minOut THEN
     #statOutput := #minOut;
     #minReached := True;
   ELSE
     #minReached := False;
   END_IF;

   #output := #statOutput;
END_FUNCTION_BLOCK

// ===== library: MasterCopy "LSim_PT3" =====

FUNCTION_BLOCK "LSim_PT3"   // FB54, SCL
{ S7_Optimized_Access := 'TRUE' }
VERSION : 2.01
   VAR_INPUT
      input : Real;   // input variable
      tmLag1 : Real := 29.0;   // time lag 1 in s
      tmLag2 : Real := 17.5;   // time lag 2 in s
      tmLag3 : Real := 3.1;   // time lag 3 in s
      gain : Real := 1.0;   // proportional gain
      disturb : Real;   // disturbance variable (additional to "input")
      cycle : Real := 0.1;   // sample time [in sec]
      reset : Bool;   // complete restart (#output = #input)
   END_VAR
   VAR_OUTPUT
      error : Bool;   // error (#tmLag1 <= 0 or #tmLag2 <= 0 or #tmLag3 <= 0)
      status : Word;   // status (if #error = TRUE then status = 16#8001)
      output : Real;   // output signal (if #error = FALSE)
   END_VAR
   VAR
      statFback1 : Real;   // feedback path value 1
      statFback2 : Real;   // feedback path value 2
      statFback3 : Real;   // feedback path value 3
   END_VAR
   VAR_TEMP
      tempHvar : Real;   // help variable
      tempCycleR : Real;   // cycle to real
      tempTmLag1R : Real;   // time lag 1 to real
      tempTmLag2R : Real;   // time lag 2 to real
      tempTmLag3R : Real;   // time lag 3 to real
      tempOutvNew : Real;   // new output variable
   END_VAR
BEGIN
   //=============================================================================
   //SIEMENS AG
   //(c)Copyright 2017 All Rights Reserved
   //-----------------------------------------------------------------------------
   //Library:       Library for Controlled System Simulation
   //Tested with:   S7-1500 FW V2.0 / S7-1200 FW V4.2
   //Engineering:   STEP 7 V14 Upd2 (TIA Portal)
   //Restrictions:  Cyclic interrupt
   //Requirements:  memory card needed for S7-1500
   //Functionality: Simulation of an PT3-system
   //
   //                               gain
   //  F(p) = ------------------------------------------------------
   //         (tmLag1 * p + 1) * (tmLag2 * p + 1) * (tmLag3 * p + 1)
   //          
   //  Call the simulation in a cyclic interrupt with
   //  cyclic interrupt time at least = tmLag1/10!
   //-----------------------------------------------------------------------------
   //Change log table:
   //Version  Date       Expert in charge                Changes applied
   //02.00.00 03.02.2016 Siemens Industry Online Support Release (STEP 7 V13 SP1)
   //02.00.01 02.03.2017 Siemens Industry Online Support Release (STEP 7 V14)
   //=============================================================================
   // check parameter
   IF #tmLag1 <= 0 OR #tmLag2 <= 0 OR #tmLag3 <= 0 THEN
     #error := TRUE;
     #status := W#16#8001;     // Parameter Error
     #output := #input; //write output data
     #statFback1 := #input; //write static data
     #statFback2 := #input;
     #statFback3 := #input;
     RETURN;
   ELSE
     #error := FALSE;
     #status := W#16#0000;     // no error
   END_IF;

   IF #reset THEN //complete restart routine

     #output := #input;//write output data
     #statFback1 := #input;//write static data
     #statFback2 := #input;
     #statFback3 := #input;

   ELSE //cycle mode routine

     #tempCycleR  := #cycle*1000; //transform data type
     #tempTmLag1R := #tmLag1*1000;
     #tempTmLag2R := #tmLag2*1000;
     #tempTmLag3R := #tmLag3*1000;

     IF #tempCycleR * 0.5 > #tempTmLag1R THEN //limit TM_LAG1
       #tempTmLag1R := #tempCycleR * 0.5;
     END_IF;

     IF #tempCycleR * 0.5 > #tempTmLag2R THEN //limit TM_LAG2
       #tempTmLag2R := #tempCycleR * 0.5;
     END_IF;

     IF #tempCycleR * 0.5 > #tempTmLag3R THEN //limit TM_LAG2
       #tempTmLag3R := #tempCycleR * 0.5;
     END_IF;

     //1. first order lag algorithm
     #tempHvar     := #tempCycleR / (#tempTmLag1R * 2.0); 
     #tempHvar     := (#gain * (#input + #disturb) - #statFback1) * #tempHvar / (#tempHvar + 1.0);
     #tempOutvNew  := #tempHvar + #statFback1;
     #statFback1  := #tempHvar * 2.0 + #statFback1;

     //2. first order lag algorithm
     #tempHvar     := #tempCycleR / (#tempTmLag2R * 2.0); 
     #tempHvar     := ((#tempOutvNew - #statFback2) * #tempHvar) / (#tempHvar + 1.0);
     #tempOutvNew  := #tempHvar + #statFback2;
     #statFback2  := #tempHvar * 2.0 + #statFback2;

     //3. first order lag algorithm
     #tempHvar     := #tempCycleR / (#tempTmLag3R * 2.0); 
     #tempHvar     := ((#tempOutvNew - #statFback3) * #tempHvar) / (#tempHvar + 1.0);
     #tempOutvNew  := #tempHvar + #statFback3;
     #statFback3  := #tempHvar * 2.0 + #statFback3;

     #output := #tempOutvNew; //write output

   END_IF;
END_FUNCTION_BLOCK

// ===== library: MasterCopy "LSim_PT3HeatCool" =====

FUNCTION_BLOCK "LSim_PT3HeatCool"   // FB64, SCL
{ S7_Optimized_Access := 'TRUE' }
VERSION : 2.01
   VAR_INPUT
      inputHeat : Real;   // input variable heating
      inputCool : Real;   // input variable cooling
      disturbHeat : Real;   // disturbance variable heating (additional to "inputHeat")
      disturbCool : Real;   // disturbance variable cooling (additional to "inputCool")
      ambTemp : Real := 20.0;   // ambient temperature
      gainHeat : Real := 1.5;   // proportional gain heating
      gainCool : Real := 3.0;   // proportional gain cooling
      tmLag1Heat : Real := 60.0;   // time lag 1 heating [s]
      tmLag2Heat : Real := 10.0;   // time lag 2 heating [s]
      tmLag3Heat : Real;   // time lag 3 heating [s]
      tmLag1Cool : Real := 60.0;   // time lag 1 cooling [s]
      tmLag2Cool : Real := 10.0;   // time lag 2 cooling [s]
      tmLag3Cool : Real;   // time lag 3 cooling [s]
      cycle : Real := 0.1;   // sample time [s]
   END_VAR
   VAR_OUTPUT
      output : Real;   // output variable
   END_VAR
   VAR_IN_OUT
      reset : Bool;   // complete restart
   END_VAR
   VAR
      statFback1 : Array[0..1] of Real;   // feedback value 1 heating/cooling
      statFback2 : Array[0..1] of Real;   // feedback value 2 heating/cooling
      statFback3 : Array[0..1] of Real;   // feedback value 3 heating/cooling
   END_VAR
   VAR_TEMP
      tempHvar : Real;   // helper
      tempCycleR : Real;   // sampling time
      tempTmLag1R : Real;   // delay time 1
      tempTmLag2R : Real;   // delay time 2
      tempTmLag3R : Real;   // delay time 3
      tempIndex : Int;   // control variable
      tempOutvNew : Array[0..1] of Real;   // new output value heating/cooling
   END_VAR
BEGIN
   //=============================================================================
   //SIEMENS AG
   //(c)Copyright 2017 All Rights Reserved
   //-----------------------------------------------------------------------------
   //Library:       Library for Controlled System Simulation
   //Tested with:   S7-1500 FW V2.0 / S7-1200 FW V4.2
   //Engineering:   STEP 7 V14 Upd2 (TIA Portal)
   //Restrictions:  Cyclic interrupt
   //Requirements:  memory card needed for S7-1500
   //Functionality: Simulation of an PT3-system with heating and cooling input
   //-----------------------------------------------------------------------------
   //Change log table:
   //Version  Date       Expert in charge                Changes applied
   //02.00.00 03.02.2016 Siemens Industry Online Support Release (STEP 7 V13 SP1)
   //02.00.01 02.03.2017 Siemens Industry Online Support Release (STEP 7 V14)
   //=============================================================================
   #tempOutvNew[0] := (#inputHeat + #disturbHeat) * #gainHeat;
   #tempOutvNew[1] := (#inputCool + #disturbCool) * #gainCool;

   IF #reset
   THEN
     //restart

     //write output parameters
     #output := #tempOutvNew[0] - #tempOutvNew[1] + #ambTemp;

     //write static local variables
     FOR #tempIndex := 0 TO 1 DO
       #statFback1[#tempIndex] := #tempOutvNew[#tempIndex];
       #statFback2[#tempIndex] := #statFback1[#tempIndex];
       #statFback3[#tempIndex] := #statFback2[#tempIndex];
     END_FOR;

     #reset := FALSE;
   ELSE
     //smoothing  
     #tempCycleR := #cycle;
     IF #tempCycleR < 0.001
     THEN
       //low limit sampling time
       #tempCycleR := 0.001;
     END_IF;

     FOR #tempIndex := 0 TO 1 DO

       IF #tempIndex = 0
       THEN
         #tempTmLag1R := #tmLag1Heat;
         #tempTmLag2R := #tmLag2Heat;
         #tempTmLag3R := #tmLag3Heat;
       ELSE
         #tempTmLag1R := #tmLag1Cool;
         #tempTmLag2R := #tmLag2Cool;
         #tempTmLag3R := #tmLag3Cool;
       END_IF;

       //1.delay
       IF #tempTmLag1R >= #tempCycleR * 0.5
       THEN
         #tempHvar := #tempCycleR / (2.0 * #tempTmLag1R + #tempCycleR);
         #tempHvar := (#tempOutvNew[#tempIndex] - #statFback1[#tempIndex]) * #tempHvar;
         //calculate new output value
         #tempOutvNew[#tempIndex] := #statFback1[#tempIndex] + #tempHvar;
         //calculate new feedback value
         #statFback1[#tempIndex] := #statFback1[#tempIndex] + 2.0 * #tempHvar;
       ELSE  //----------------------------------- implicit PT1
         #tempHvar := #tempCycleR / (#tempTmLag1R + #tempCycleR);
         //calculate new feedback value
         #statFback1[#tempIndex] := #statFback1[#tempIndex] + (#tempOutvNew[#tempIndex] - #statFback1[#tempIndex]) * #tempHvar;
         //calculate new output value
         #tempOutvNew[#tempIndex] := #statFback1[#tempIndex];
       END_IF;

       //2.delay heating
       IF #tempTmLag2R >= #tempCycleR * 0.5
       THEN
         #tempHvar := #tempCycleR / (2.0 * #tempTmLag2R + #tempCycleR);
         #tempHvar := (#tempOutvNew[#tempIndex] - #statFback2[#tempIndex]) * #tempHvar;
         //calculate new output value
         #tempOutvNew[#tempIndex] := #statFback2[#tempIndex] + #tempHvar;
         //calculate new feedback value
         #statFback2[#tempIndex] := #statFback2[#tempIndex] + 2.0 * #tempHvar;
       ELSE
         #statFback2[#tempIndex] := #tempOutvNew[#tempIndex];
       END_IF;

       //3.delay heating
       IF #tempTmLag3R >= #tempCycleR * 0.5
       THEN
         #tempHvar := #tempCycleR / (2.0 * #tempTmLag3R + #tempCycleR);
         #tempHvar := (#tempOutvNew[#tempIndex] - #statFback3[#tempIndex]) * #tempHvar;
         //calculate new output value
         #tempOutvNew[#tempIndex] := #statFback3[#tempIndex] + #tempHvar;
         //calculate new feedback value
         #statFback3[#tempIndex] := #statFback3[#tempIndex] + 2.0 * #tempHvar;
       ELSE
         #statFback3[#tempIndex] := #tempOutvNew[#tempIndex];
       END_IF;

     END_FOR;

     #output := #tempOutvNew[0] - #tempOutvNew[1] + #ambTemp;
   END_IF;
END_FUNCTION_BLOCK

// ===== library: MasterCopy "LSim_TempProcess" =====

FUNCTION_BLOCK "LSim_TempProcess"   // FB58, SCL
{ S7_Optimized_Access := 'TRUE' }
VERSION : 2.01
   VAR_INPUT
      inTemp : Real;   // Temperature Input [K] ("useHeatPow" must be FALSE to use this input)
      useHeatPow : Bool := TRUE;   // Use "heatPow" as input
      activHeatPow : Bool;   // Turn on heating ("useHeatPow" must be TRUE to use this input)
      activCoolRth : Bool;   // Turn on cooling by "statRThCool"
      activCoolPow : Bool;   // Turn on cooling by "coolPow"
      coolPow : Real;   // Positive value of energy reduction caused by succeding process [W]
      ambTemp : Real := 20.0;   // Ambient Temperature in °C
      cycle : Real := 0.1;   // Call cycle time in s
      reset : Bool;   // Reset internal variables
   END_VAR
   VAR_OUTPUT
      outTemp : Real;   // [°C]
      interTemp : Real;   // [°C]
   END_VAR
   VAR_IN_OUT
      heatPow : Real;   // Heater Energy in [W]
   END_VAR
   VAR
      statRthTrans1 : Real := 1.5;   // Input thermal resistance in transition to capacitor 1 [K/W]
      statRth1 : Real := 1.0;   // Thermal resistance parallel to thermal capacity 1 [K/W]
      statRthTrans2 : Real := 1.5;   // Thermal resistance for energy transition from capacity 1 to capacity 2 [K/W]
      statRth2 : Real := 1.0;   // Thermal resistance parallel to thermal capacity 2 [K/W]
      statRthCool : Real := 2.0;   // Thermal resistance of cooling device [K/W]
      statCth1 : Real := 10.0;   // Thermal Capacity 1 [Ws/K]
      statCth2 : Real := 30.0;   // Thermal Capacity 2 [Ws/K]
      statZInt1 : Real;   // internal
      statZInt2 : Real;   // internal
      statUc1 : Real;   // internal
      statUc2 : Real;   // internal
      statIth2 : Real;   // internal
   END_VAR
   VAR_TEMP
      tempSumPoint1 : Real;
      tempSumPoint2 : Real;
   END_VAR
BEGIN
   //=============================================================================
   //SIEMENS AG
   //(c)Copyright 2017 All Rights Reserved
   //-----------------------------------------------------------------------------
   //Library:       Library for Controlled System Simulation
   //Tested with:   S7-1500 FW V2.0 / S7-1200 FW V4.2
   //Engineering:   STEP 7 V14 Upd2 (TIA Portal)
   //Restrictions:  Cyclic interrupt
   //Requirements:  memory card needed for S7-1500
   //Functionality: Simulates of an asymmetrical temperature process which can be
   //actively heated and cooled down (also passively).
   //-----------------------------------------------------------------------------
   //Change log table:
   //Version  Date       Expert in charge                Changes applied
   //02.00.00 03.02.2016 Siemens Industry Online Support Release (STEP 7 V13 SP1)
   //02.00.01 02.03.2017 Siemens Industry Online Support Release (STEP 7 V14)
   //=============================================================================
   IF #reset = TRUE THEN
     // Reset all variables
     #statUc1 := 0;
     #statUc2 := 0;
     #statIth2 := 0;
     #tempSumPoint1 := 0;
     #tempSumPoint2 := 0;
     #statZInt1 := 0;
     #statZInt2 := 0;
   END_IF;

   IF #useHeatPow = FALSE THEN
     // Temperature Input will be used, so "heatPow" will be used as output
     #heatPow := ((#inTemp - #ambTemp - #statUc1) / #statRthTrans1);
   END_IF;

   // Calculate fist summing point
   IF (#activHeatPow = TRUE) OR (#useHeatPow = FALSE) THEN
     #tempSumPoint1 := #heatPow - (#statUc1 / #statRth1) - #statIth2;
   ELSE
     #tempSumPoint1 := 0 - (#statUc1 / #statRth1) - #statIth2;
   END_IF;

   // Calculate integrator 1
   #statUc1 := #statUc1 + (((#tempSumPoint1 / #statCth1) + #statZInt1) * #cycle * 0.5);
   #statZInt1 := #tempSumPoint1 / #statCth1;

   // Calculate intermidiate temperature
   #interTemp := #statUc1 + #ambTemp;

   // Calculate thermal power flow from Integrator 1 to Integrator 2
   #statIth2 := ((#statUc1 - #statUc2) / #statRthTrans2);

   // Calculate summing point 2
   IF #activCoolPow = TRUE THEN
     #tempSumPoint2 := #statIth2 - (#statUc2 / #statRth2) - #coolPow;
   ELSE
     #tempSumPoint2 := #statIth2 - (#statUc2 / #statRth2);
   END_IF;

   IF #activCoolRth = TRUE THEN
     // Cooling is activated
     #tempSumPoint2 := #tempSumPoint2 - (#statUc2 / #statRthCool);
   END_IF;

   // Calculate Integrator 2
   #statUc2 := (#cycle * 0.5 * ((#tempSumPoint2 / #statCth2) + #statZInt2)) + #statUc2;
   #statZInt2 := #tempSumPoint2 / #statCth2;

   // Calculate Output Temperature
   #outTemp := #statUc2 + #ambTemp;
END_FUNCTION_BLOCK

// ===== library: MasterCopy "LSim_Valve" =====

FUNCTION_BLOCK "LSim_Valve"   // FB63, FBD
{ S7_Optimized_Access := 'TRUE' }
VERSION : 2.01
// //============================================================================
// //SIEMENS AG
// //(c)Copyright 2017 All Rights Reserved
// //-----------------------------------------------------------------------------
// //Library:       Library for Controlled System Simulation
// //Tested with:   S7-1500 FW V2.0 / S7-1200 FW V4.2
// //Engineering:   STEP 7 V14 Upd2 (TIA Portal)
// //Restrictions:  Cyclic interrupt
// //Requirements:  memory card needed for S7-1500
// //Functionality: Simulation of a valve with adjustable transition time
// //-----------------------------------------------------------------------------
// //Change log table:
// //Version    Date             Expert in charge                               Changes applied
// //02.00.00 03.02.2016 Siemens Industry Online Support Release (STEP 7 V13 SP1)
// //02.00.01 02.03.2017 Siemens Industry Online Support Release (STEP 7 V14)
// //============================================================================
   VAR_INPUT
      inputUp : Bool := false;   // control signal “Open valve”
      inputDn : Bool := false;   // control signal “Close valve”
      inputPer : Int;   // Analog manipulated variable
      perOn : Bool;   // selection switch, whether inputUp/inputDn or inputPer is used (inputPer is used for TRUE)
      perMax : Real := 27648.0;   // upper limit of the analog value of the valve position.
      perMin : Real;   // lower limit of the analog value of the valve position
      realMax : Real := 100.0;   // upper limit of the converted floating-point value for the valve position
      realMin : Real;   // lower limit of the converted floating-point value for the valve position
      transitTime : Real := 20.0;   // traversing time of the value between the end positions
      cycle : Real := 0.1;   // cyclic time [sec]
      reset : Bool := false;   // resets all relevant parameters to ‘0’ including the output
   END_VAR
   VAR_OUTPUT
      output : Real := 0.0;   // calculated valve position (within the “realMin” and “realMax” limits)
      outputPer : Int;   // calculated analog valve position (within the “perMin” and “perMax” limits)
      highLimit : Bool := false;   // simulated upper valve end position reached at highLimit = TRUE
      lowLimit : Bool := false;   // simulated lower valve end position reached at lowLimit = TRUE
   END_VAR
   VAR
      statInput : Real;
      statDelta : Real;
      statOut : Real;
      statHigh : Bool;
      statLow : Bool;
   END_VAR
   VAR_TEMP
      tempReal : Real;
      tempStepWidth : Real;
      tempStepWidthNeg : Real;
      tempBool : Bool;
      tempInputNorm : Real;
      tempUpFlag : Bool;
      tempDnFlag : Bool;
      tempInt : Int;
   END_VAR
   VAR_TEMP   // added for the SCL form of the ladder/FBD networks
      _w1 : Bool;
   END_VAR
BEGIN

REGION Network 1: reset
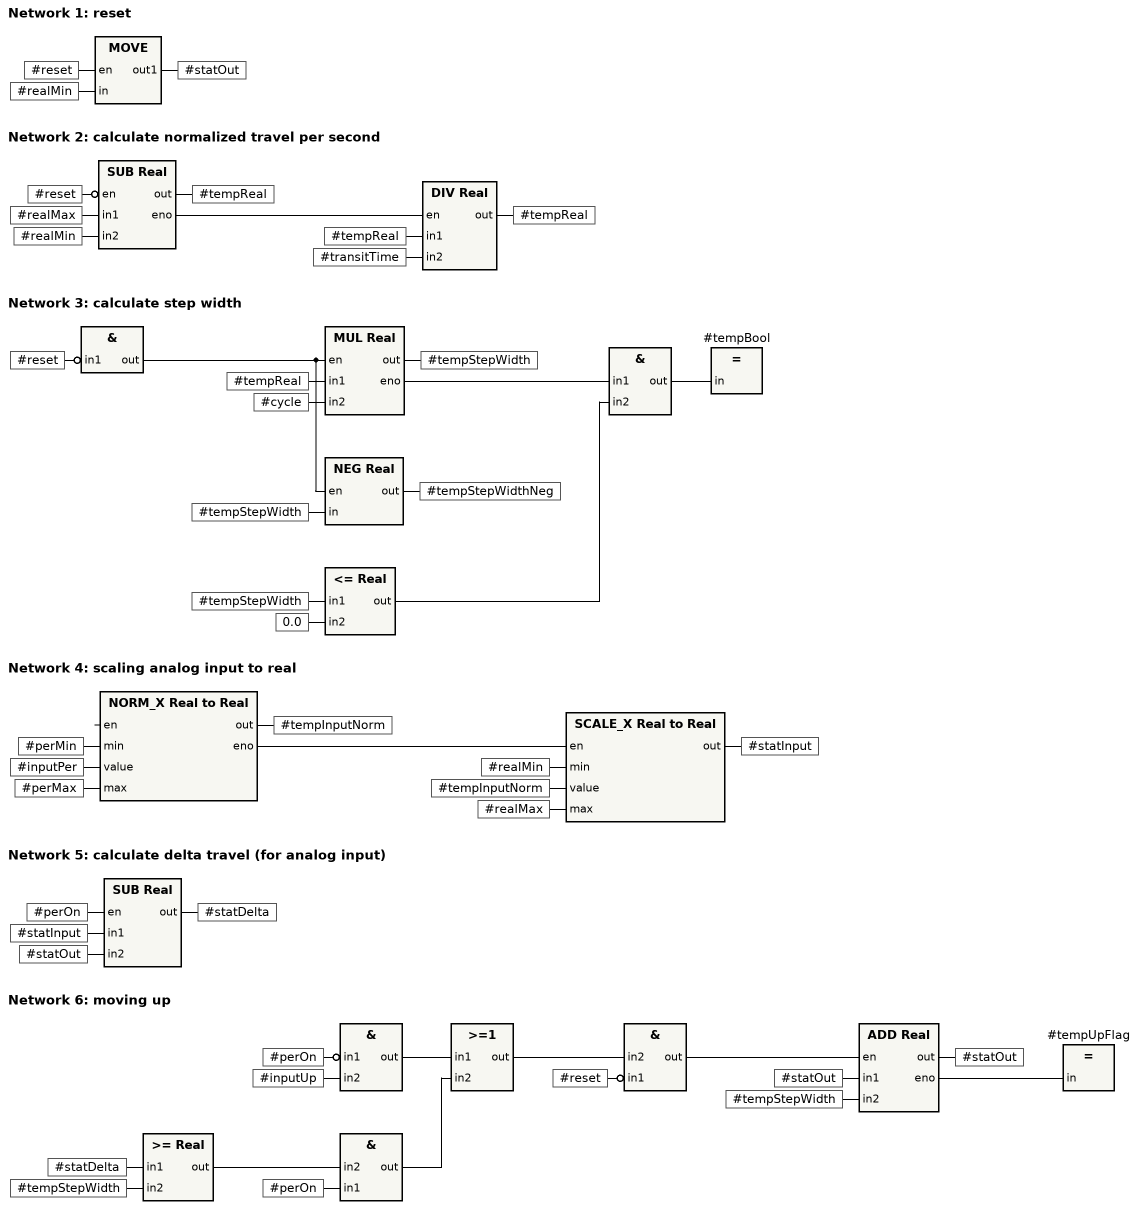
   IF #reset THEN #statOut := #realMin; END_IF;
END_REGION

REGION Network 2: calculate normalized travel per second
   // ENO of a box is taken as its EN; it also drops when the box reports an error
   IF NOT #reset THEN
       #tempReal := #realMax - #realMin;
       #tempReal := #tempReal / #transitTime;
   END_IF;
END_REGION

REGION Network 3: calculate step width
   // ENO of a box is taken as its EN; it also drops when the box reports an error
   IF NOT #reset THEN #tempStepWidth := #tempReal * #cycle; END_IF;
   #tempBool := NOT #reset AND (#tempStepWidth <= 0.0);
   IF NOT #reset THEN #tempStepWidthNeg := -#tempStepWidth; END_IF;
END_REGION

REGION Network 4: scaling analog input to real
   // ENO of a box is taken as its EN; it also drops when the box reports an error
   #tempInputNorm := NORM_X(MIN := #perMin, VALUE := #inputPer, MAX := #perMax);
   #statInput := SCALE_X(MIN := #realMin, VALUE := #tempInputNorm, MAX := #realMax);
END_REGION

REGION Network 5: calculate delta travel (for analog input)
   IF #perOn THEN #statDelta := #statInput - #statOut; END_IF;
END_REGION

REGION Network 6: moving up
   // ENO of a box is taken as its EN; it also drops when the box reports an error
   #_w1 := ((NOT #perOn AND #inputUp) OR ((#statDelta >= #tempStepWidth) AND #perOn)) AND NOT #reset;
   IF #_w1 THEN #statOut := #statOut + #tempStepWidth; END_IF;
   #tempUpFlag := #_w1;
END_REGION

REGION Network 7: checking max. limit
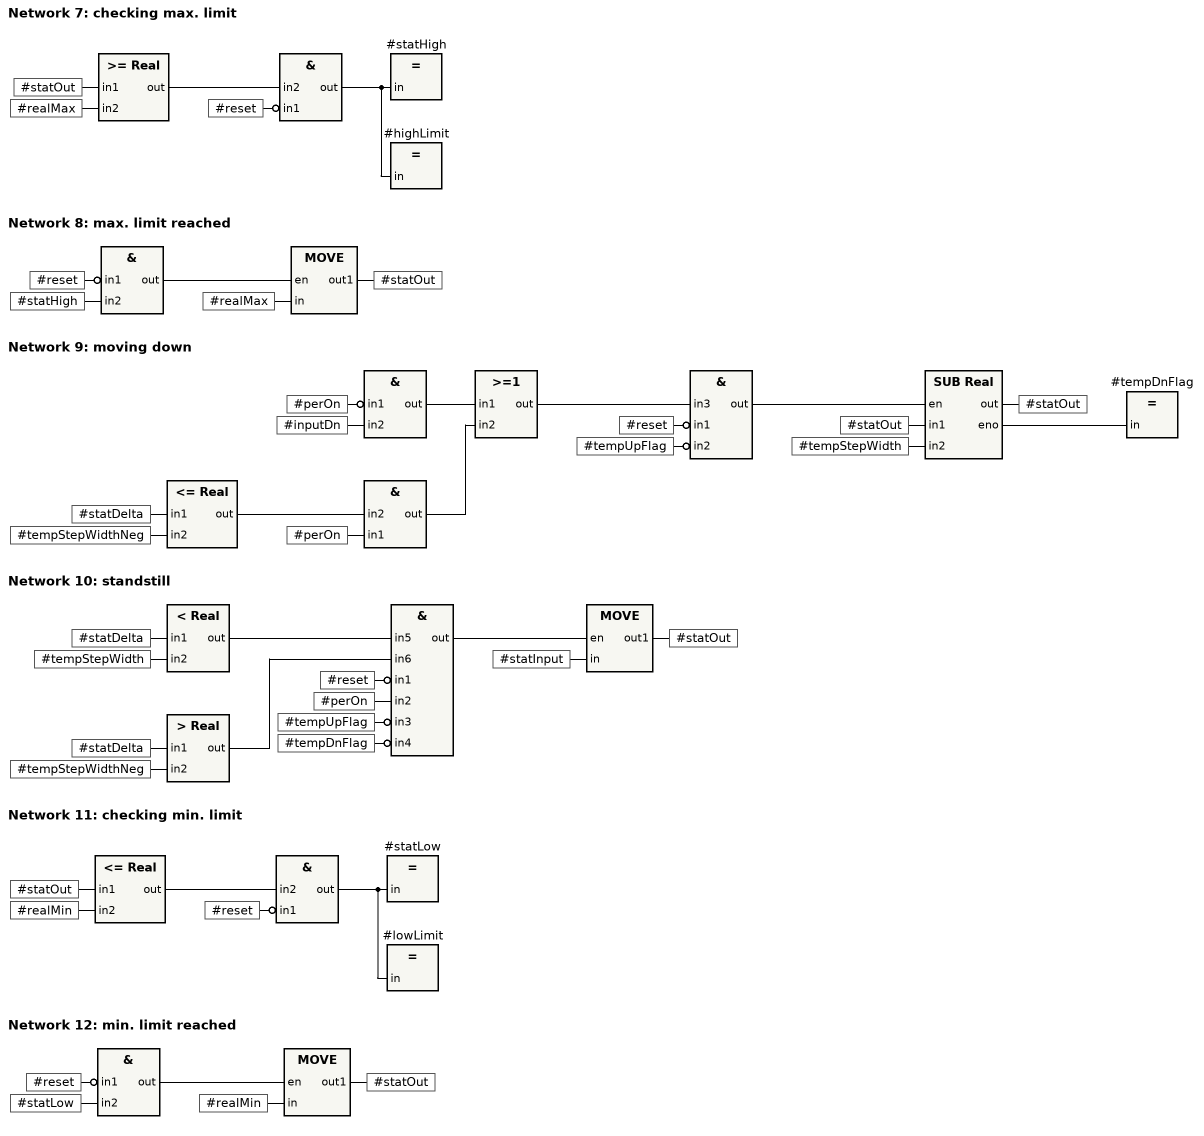
   #statHigh := (#statOut >= #realMax) AND NOT #reset;
   #highLimit := #statHigh;
END_REGION

REGION Network 8: max. limit reached
   IF NOT #reset AND #statHigh THEN #statOut := #realMax; END_IF;
END_REGION

REGION Network 9: moving down
   // ENO of a box is taken as its EN; it also drops when the box reports an error
   #_w1 := ((NOT #perOn AND #inputDn) OR ((#statDelta <= #tempStepWidthNeg) AND #perOn)) AND NOT #reset AND NOT #tempUpFlag;
   IF #_w1 THEN #statOut := #statOut - #tempStepWidth; END_IF;
   #tempDnFlag := #_w1;
END_REGION

REGION Network 10: standstill
   IF (#statDelta < #tempStepWidth) AND (#statDelta > #tempStepWidthNeg) AND NOT #reset AND #perOn AND NOT #tempUpFlag AND NOT #tempDnFlag THEN
       #statOut := #statInput;
   END_IF;
END_REGION

REGION Network 11: checking min. limit
   #statLow := (#statOut <= #realMin) AND NOT #reset;
   #lowLimit := #statLow;
END_REGION

REGION Network 12: min. limit reached
   IF NOT #reset AND #statLow THEN #statOut := #realMin; END_IF;
END_REGION

REGION Network 13: output and scaling to analog
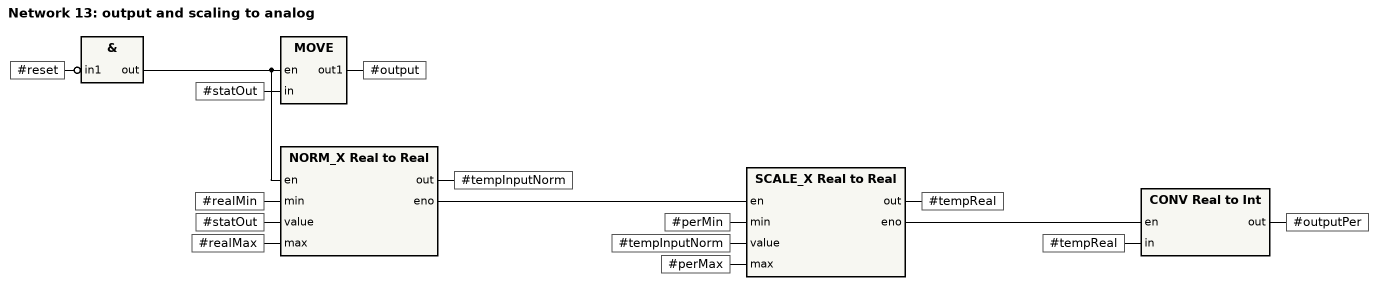
   // ENO of a box is taken as its EN; it also drops when the box reports an error
   IF NOT #reset THEN
       #output := #statOut;
       #tempInputNorm := NORM_X(MIN := #realMin, VALUE := #statOut, MAX := #realMax);
       #tempReal := SCALE_X(MIN := #perMin, VALUE := #tempInputNorm, MAX := #perMax);
       #outputPer := REAL_TO_INT(#tempReal);
   END_IF;
END_REGION
END_FUNCTION_BLOCK

// ===== library: MasterCopy "LSim_Multizone" =====

FUNCTION_BLOCK "LSim_Multizone"   // FB65, SCL
{ S7_Optimized_Access := 'TRUE' }
VERSION : 1.1
   VAR_INPUT
      ambTemp : Real := 20.0;   // Ambient temperature
      reset : Bool;   // Reset block
      cycle : Real := 0.1;   // Cyclic interrupt time in seconds
   END_VAR
   VAR_OUTPUT
      error : Bool;   // Error occurred (block stopped working)
      statusID : UInt;   // Error source (see comment)
      status : Word;   // Error code (see comment)
      maxReached : Bool;   // Output of "LSim_PT1" or "LSim_PT2aper" has reached max. limit
      minReached : Bool;   // Output of "LSim_PT1" or "LSim_PT2aper" has reached min. limit
   END_VAR
   VAR_IN_OUT
      zones : Array[1..#MAX] of "LSim_typeZone";   // Zone parameters
   END_VAR
   VAR
      statZ : Array[1..#MAX] of "LSim_typeDynState";   // Internal parameters for calculation
      instPT2Z : Array[1..#MAX] of "LSim_PT2aper";   // LSim_PT2aper instances
      instHeatZ : Array[1..#MAX] of "LSim_PT1";   // LSim_PT1 instances for heating
      instCoolZ : Array[1..#MAX] of "LSim_PT1";   // LSim_PT1 instances for cooling
   END_VAR
   VAR_TEMP
      tempIndex : DInt;
   END_VAR
   VAR CONSTANT
      MAX : DInt := 3;   // Numbers of zones
      TMLAG_HEATER : Real := 5.0;   // Time constant for PT1 (heating)
      TMLAG_COOLER : Real := 10.0;   // Time constant for PT1 (cooling)
      GAIN_ZONE : Real := 5.0;   // Gain factor for PT2 (temperature)
      TMLAG1_ZONE : Real := 20.0;   // Time constant 1 for PT2 (temperature)
      TMLAG2_ZONE : Real := 3.0;   // Time constant 2 for PT2 (temperature)
      PT2_MAX_OUT : Real := 1000.0;   // Maximum output limit for PT2 (temperature)
      PT2_MIN_OUT : Real := -1000.0;   // Minimum output limit for PT2 (temperature)
   END_VAR
BEGIN
   //=============================================================================
   //SIEMENS AG
   //(c)Copyright 2017 All Rights Reserved
   //-----------------------------------------------------------------------------
   //Library:       Library for Controlled System Simulation
   //Tested with:   S7-1500 FW V2.0 / S7-1200 FW V4.2
   //Engineering:   STEP 7 V14 Upd2 (TIA Portal)
   //Restrictions:  Cyclic interrupt
   //Requirements:  SIMATIC Memory Card for using S7-1500 CPU
   //Functionality: Simple simulation of coupled thermal zones
   //---------------------------------------------------------------------
   //Change log table:
   //Version  Date       Expert in charge                Changes applied
   //01.00.00 12.10.2016 Siemens Industry Online Support Release (STEP 7 V14)
   //01.00.01 06.03.2017 Siemens Industry Online Support Release in LSim
   //=====================================================================
   // Inputs:
   //              heating and cooling input (0..100%) for all zones via
   //              #zones[X].inputHeat,
   //              #zones[X].inputCool and
   //              #zones[X].disturbance
   // Outputs:
   //              the simulated temperatur for all zones via
   //              #zones[X].output
   // Error handling:
   //              error source #statusID = z*10 + n*1; z =zone
   //              n = 1: FB "LSim_PT1" (instHeatZ[z])
   //              n = 2: FB "LSim_PT1" (instCoolZ[z])
   //              n = 3: FB "LSim_PT2aper" (instPT2Z[z])
   //              
   //              Example: #statusID = 21
   //              ->  error source: FB "LSim_PT1" (instHeatZ[2])
   //              
   //              error code #status
   //              -> see comment #status of error source
   //=====================================================================

   REGION PT1 
     FOR #tempIndex := 1 TO #MAX DO
       // Simulation of Heating and Cooling actuator logic for each thermal zone

       REGION heat
         // Zone Heater dynamics (PT1) 0..100%, tmLag1 = 5sek
         #instHeatZ[#tempIndex]instHeatZ(input := #zones[#tempIndex].inputHeat,
                                tmLag1 := #TMLAG_HEATER,
                                cycle := #cycle,
                                reset := #reset);

         IF (#instHeatZ[#tempIndex].error = TRUE) THEN
           #error := TRUE;
           #statusID := 10 * DINT_TO_UINT(#tempIndex) + 1;
           #status := #instHeatZ[#tempIndex].status;
           RETURN;
         END_IF;
       END_REGION

       REGION cool
         // Zone Cooler dynamics (PT1) 0.100%, tmLag1 = 10sek
         #instCoolZ[#tempIndex]instCoolZ(input := #zones[#tempIndex].inputCool,
                                tmLag1 := #TMLAG_COOLER,
                                cycle := #cycle,
                                reset := #reset);

         IF (#instCoolZ[#tempIndex].error = TRUE) THEN
           #error := TRUE;
           #statusID := 10 * DINT_TO_UINT(#tempIndex) + 2;
           #status := #instCoolZ[#tempIndex].status;
           RETURN;
         END_IF;
       END_REGION
       // generate input variable for thermal simulation area zone
       #statZ[#tempIndex].uInp := #instHeatZ[#tempIndex].output
       - #instCoolZ[#tempIndex].output
       + #zones[#tempIndex].disturbance;

     END_FOR;
   END_REGION

   REGION coupling
     //===================================================================================
     // dynamic simulation of at least 3 thermal coupled zones
     // Connection logic between thermal zones
     //===================================================================================

     //First zone: previous zone doesn't exist -> (#statZ[z-1].y * #statZ[z-1].kFor)= 0
     #statZ[1].u := #statZ[1].uInp
     - (2 * (#statZ[1].y * #statZ[1].kInt))
     + (#statZ[2].y * #statZ[2].kBack);

     FOR #tempIndex := 2 TO (#MAX - 1) DO
       // 1 < zone < max: #statZ[z].u := #statZ[z].uInp
       // + (#statZ[z-1].y * #statZ[z-1].kFor)
       // - (2 * (#statZ[z].y * #statZ[z].kint))
       // + (#statZ[z+1].y * #statZ[z+1].kBack);
       #statZ[#tempIndex].u := #statZ[#tempIndex].uInp
       + (#statZ[(#tempIndex - 1)].y * #statZ[(#tempIndex - 1)].kFor)
       - (2 * (#statZ[#tempIndex].y * #statZ[#tempIndex].kInt))
       + (#statZ[(#tempIndex + 1)].y * #statZ[(#tempIndex + 1)].kBack);
     END_FOR;

     //Last zone: next Zone doesn't exist -> (#statZ[z+1].y * #statZ[z+1].kBack);)= 0
     #statZ[#MAX].u := #statZ[#MAX].uInp
     + (#statZ[(#MAX - 1)].y * #statZ[(#MAX - 1)].kFor)
     - (2 * (#statZ[#MAX].y * #statZ[#MAX].kInt));
   END_REGION

   REGION PT2
     FOR #tempIndex := 1 TO #MAX DO
       // dynamic Simulation of zone (PT2)
       #instPT2Z[#tempIndex]instPT2Z(input := #statZ[#tempIndex].u,
                             tmLag1 := #TMLAG1_ZONE,
                             tmLag2 := #TMLAG2_ZONE,
                             gain := #GAIN_ZONE,
                             cycle := #cycle,
                             maxOut := #PT2_MAX_OUT,
                             minOut := #PT2_MIN_OUT,
                             reset := #reset,
                             output => #statZ[#tempIndex].y);

       IF (#instPT2Z[#tempIndex].error = TRUE) THEN
         #error := TRUE;
         #statusID := 10 * DINT_TO_UINT(#tempIndex) + 3;
         #status := #instPT2Z[#tempIndex].status;
         RETURN;
       END_IF;

       // Output of simulation model adding ambient temperature
       #zones[#tempIndex].output := #statZ[#tempIndex].y + #ambTemp;

     END_FOR;
   END_REGION

   FOR #tempIndex := 1 TO #MAX DO
     //Reached handling (PT1 & PT2)
     IF #instHeatZ[#tempIndex].maxReached OR #instCoolZ[#tempIndex].maxReached OR #instPT2Z[#tempIndex].maxReached THEN
       #maxReached := TRUE;
     END_IF;

     IF #instHeatZ[#tempIndex].minReached OR #instCoolZ[#tempIndex].minReached OR #instPT2Z[#tempIndex].minReached THEN
       #minReached := TRUE;
     END_IF;

   END_FOR;

   IF (#reset = TRUE) THEN
     #maxReached := FALSE;
     #minReached := FALSE;
   END_IF;
END_FUNCTION_BLOCK

// ===== library: MasterCopy "LSim_typeDynState" =====

TYPE "LSim_typeDynState"
// V1.1
   STRUCT
      kInt : Real := 0.2;   // coupling constant internal
      kFor : Real := 0.3;   // coupling constant forwards
      kBack : Real := 0.1;   // coupling constant backwards
      uInp : Real;   // uInp = heatPT1out - coolPT1out + disturbance
      u : Real;   // u = uInp + kFor(z-1) * y(z-1) - 2 * kInt * y + kBack(z+1) * y(z+1); z = zone
      y : Real;   // y = PT2out
   END_STRUCT;
END_TYPE

// ===== library: MasterCopy "LSim_typeZone" =====

TYPE "LSim_typeZone"
// V1.1
   STRUCT
      inputHeat : Real;   // input value in REAL format - heating / Ausgangswert im REAL-Format - Heizen
      inputCool : Real;   // input value in REAL format - cooling / Ausgangswert im REAL-Format - Kühlen
      disturbance : Real;   // disturbance (input)
      output : Real;   // zone temperature (output)
   END_STRUCT;
END_TYPE